(********************* G.D S.p.A. - Technical Department ***********************************
This program has been generated automatically from Application Designer DE&F
********************************************************************************************)
PROGRAM dbg_csp_transfer_infeed_reject_highload
VAR
  high_achk_shd : analog_check_shadow;
  high_ai_shd : analog_input_shadow;
END_VAR

_objects_manager();

IF	g_application_status <> APPLICATION_STATUS_RUNNING
THEN
	RETURN;
END_IF

CASE process_get_mode(CONVERSION_this := dbg_root.prc) OF
	MODE_ABSENT,
	MODE_INACTIVE:
		RETURN;
	MODE_TEST:
		RETURN;
END_CASE

ACTION _objects_manager:
IF	objects_initialization()
THEN
	analog_check_shadow_init(
		sim_mode:= SHADOW_SIMULATION_MODE_AUTOMATIC, 
		father:= csp_transfer_infeed_reject_highload.high_achk, 
		process:= dbg_root.prc, 
		CONVERSION_this:= high_achk_shd);

	analog_input_shadow_init(
		sim_mode:= SHADOW_SIMULATION_MODE_AUTOMATIC, 
		father:= csp_transfer_infeed_reject_highload.high_ai, 
		process:= dbg_root.prc, 
		CONVERSION_this:= high_ai_shd);

	RETURN;
END_IF

IF	objects_running()
THEN
	analog_check_shadow_cycle(high_achk_shd);
	analog_input_shadow_cycle(high_ai_shd);
END_IF
END_ACTION

END_PROGRAM

(* stored: Version 1.1.0.1, ProductVersion 3.1.4022.12
   POU dbg_csp_transfer_infeed_reject_highload: Id {51ea3052-5716-4867-8a27-1d58a3613020}, SpecialFunc None
   Action _objects_manager: Id {7eead544-be7d-4e6d-ac7c-6b9c6e0306b7} *)
